{attribute 'reflection'} 
(* The VLT® PROFINET MCA 120 is used in combination with:
• VLT® HVAC Drive FC 102
• VLT® Refrigeration Drive FC 103
• VLT® AQUA Drive FC 202
• VLT® AutomationDrive FC 301/302
• VLT® Decentral Drive FCD 302
 *)
FUNCTION_BLOCK FB_Danfoss_VLT_MCA_120 EXTENDS FB_LinkDataReal
VAR_INPUT	
	stControl				: ST_Danfoss_VLT_MCA_120_Control;	
	stConfig 				: ST_Danfoss_VLT_MCA_120_Config;
END_VAR

VAR_OUTPUT
	stStatus				: ST_Danfoss_VLT_MCA_120_Status;
	fValue					: REAL;
END_VAR

VAR
    {attribute 'instance-path'} 
    {attribute 'noinit'} 
    sPath 					: STRING; 
	pFromBus				: POINTER TO BYTE;
	pToBus					: POINTER TO BYTE;	
	                    	
	fbProfidriveGSM			: FB_ProfidriveGSM;	
	fbMoveVelocity			: FB_MoveVelocity;
	
	fAcceleration	 		: REAL;
	fDeceleration		 	: REAL;
	fDecelerationQuickStop 	: REAL;
	fDecelerationCoastStop 	: REAL;
	bQuickStopExternal		: BOOL;
	
	bFaultPresent 			: BOOL;
	bAlarmPresent 			: BOOL;
	bInverterError 			: BOOL;
	bVoltageError 			: BOOL;
	bMomentError 			: BOOL;
	bTimerError 			: BOOL;
END_VAR

SUPER^();
InitRun();
ReadBus();
ControlLogic();
WriteBus();

(*Assign Process Data Objects to device*)
METHOD PUBLIC AssignProcessData : BOOL
VAR_INPUT
	aControlData 		: ANY; //Addr. Process Output (PO), 6 BYTES FROM FIELDBUS
	aStatusData 		: ANY; //Addr. Process Input (PI), 6 BYTES TO FIELDBUS
END_VAR
THIS^.pFromBus := aControlData.pValue;
THIS^.pToBus := aStatusData.pValue;
END_METHOD

METHOD INTERNAL ControlLogic
(* Evaluate/limit parameters *)
	EvaluateParameters();

(* Unity init - load position *)
	IF SUPER^.Status.7 THEN
		ControlData := StatusData;
	END_IF

(* Call base statemachine *)
fbProfidriveGSM.bStandstill						:= OC_Core.F_Compare(fbMoveVelocity.fVelocity, 0, 1E-3);
fbProfidriveGSM.stControl.b0_On 				:= stControl.bOFF1;
fbProfidriveGSM.stControl.b1_CoastStop 			:= stControl.bOFF2;
fbProfidriveGSM.stControl.b2_QuickStop 			:= stControl.bOFF3 AND NOT bQuickStopExternal;
fbProfidriveGSM.stControl.b3_EnableOperation	:= stControl.bEnableOperation;

(* Preset target values *)
	fbMoveVelocity.fTargetVelocity	:= 0;
	fbMoveVelocity.fAccMax 			:= fAcceleration;
	fbMoveVelocity.fDecMax 			:= fDeceleration;

(* Operation *)
	IF fbProfidriveGSM.eState = E_ProfidriveGSM_State.S4_Operation THEN	
		// Main setpoint
		IF NOT stControl.bJog1 AND NOT stControl.bJog2 THEN
			fbMoveVelocity.fTargetVelocity := (stControl.nSoll * stConfig.fP2000) / 16#4000;
		// Jog 1
		ELSIF stControl.bJog1 AND NOT stControl.bJog2 THEN
			fbMoveVelocity.fTargetVelocity := stConfig.fP1058;
		// Jog 2
		ELSIF NOT stControl.bJog1 AND stControl.bJog2 THEN	
			fbMoveVelocity.fTargetVelocity := stConfig.fP1059;
		END_IF
		
		// Stop
		IF NOT stControl.bOperatingCondition OR NOT stControl.bEnableSetpoint THEN
			fbMoveVelocity.fTargetVelocity := 0;
		END_IF
		
		// Reversing velocity
		IF stControl.bReversing THEN
			fbMoveVelocity.fTargetVelocity := -fbMoveVelocity.fTargetVelocity;
		END_IF
		
		// Hold velocity
		IF NOT stControl.bContinueRampFunctionGenerator AND NOT stControl.bJog1 AND NOT stControl.bJog2 THEN
			fbMoveVelocity.fTargetVelocity := fbMoveVelocity.fVelocity;
		END_IF	
		
	END_IF
	
(* Coast stop, Quick stop, Ramp stop *)
	IF fbProfidriveGSM.eState = E_ProfidriveGSM_State.S1_SwitchingOnInhibited THEN
		fbMoveVelocity.fTargetVelocity	:= 0;
		fbMoveVelocity.fAccMax 			:= fDecelerationCoastStop;
		fbMoveVelocity.fDecMax 			:= fDecelerationCoastStop;
	ELSIF fbProfidriveGSM.eState = E_ProfidriveGSM_State.S52_QuickStop THEN
		fbMoveVelocity.fTargetVelocity	:= 0;
		fbMoveVelocity.fAccMax 			:= fDecelerationQuickStop;
		fbMoveVelocity.fDecMax 			:= fDecelerationQuickStop;
	ELSIF fbProfidriveGSM.eState = E_ProfidriveGSM_State.S51_RampStop THEN
		fbMoveVelocity.fTargetVelocity	:= 0;
		fbMoveVelocity.fAccMax 			:= fDeceleration;
		fbMoveVelocity.fDecMax 			:= fDeceleration;
	END_IF

(* Call MoveVelocity *)
	fbMoveVelocity();
	
(* Status word *)
	stStatus.bReadyForSwitchingOn			:= fbProfidriveGSM.stStatus.b0_ReadyToSwitchOn;	
	stStatus.bReadyForOperation				:= fbProfidriveGSM.stStatus.b1_ReadyForOperation;
	stStatus.bOperationEnabled				:= stControl.bEnableOperation;
	stStatus.bFaultPresent					:= bFaultPresent;
	stStatus.bNoCoastDownActive				:= fbProfidriveGSM.eState <> E_ProfidriveGSM_State.S1_SwitchingOnInhibited;
	stStatus.bNoQuickStopActive				:= fbProfidriveGSM.eState <> E_ProfidriveGSM_State.S52_QuickStop;
	stStatus.bSwitchingOnInhibited			:= fbProfidriveGSM.stStatus.b6_SwitchingOnInhibited;
	stStatus.bAlarmPresent					:= bAlarmPresent;
	stStatus.bDeviationWithinTolerance		:= TRUE;
	stStatus.bControlRequested				:= stConfig.bControlRequested;	
	stStatus.bFrequencyLimitOk				:= TRUE;	
	stStatus.bBusy							:= ABS(fbMoveVelocity.fVelocity) > 0;
	stStatus.bInverterError					:= bInverterError;	
	stStatus.bVoltageError					:= bVoltageError;
	stStatus.bMomentError					:= bMomentError;
	stStatus.bTimerError					:= bTimerError;

(* Reset quickstop from extern *)
	IF stControl.bAcknowledgeFaults THEN
		bQuickStopExternal := FALSE;
	END_IF

(* Calculate NIST *)
	IF stConfig.fP2000 = 0 THEN
		stStatus.nIst	:= 0;
	ELSE
		stStatus.nIst	:=	REAL_TO_INT((ABS(fbMoveVelocity.fVelocity) * 16#4000) / stConfig.fP2000);
	END_IF

(* Output of actual value *)	
	IF stConfig.bOutputVelocity THEN
		ControlData := fbMoveVelocity.fVelocity;
	ELSE
		ControlData := ControlData + fbMoveVelocity.fVelocity *  GVL_Core.fbSystem.fDeltaTime * GVL_Core.fbSystem.fTimeScaling;
	END_IF
	
	fValue := ControlData;
END_METHOD

METHOD INTERNAL EvaluateParameters
VAR_INPUT
END_VAR
IF stConfig.fP1120 > 0 THEN
	fAcceleration := stConfig.fP2000/stConfig.fP1120;
ELSE
	fAcceleration := 1000;
END_IF

IF stConfig.fP1121 > 0 THEN
	fDeceleration := stConfig.fP2000/stConfig.fP1121;
ELSE
	fDeceleration := 1000;
END_IF

IF stConfig.fP1135 > 0 THEN
	fDecelerationQuickStop := stConfig.fP2000/stConfig.fP1135;
ELSE
	fDecelerationQuickStop := 1000;
END_IF

IF stConfig.fRampDownTimeCoastStop > 0 THEN
	fDecelerationCoastStop := stConfig.fP2000/stConfig.fRampDownTimeCoastStop;
ELSE
	fDecelerationCoastStop := 1000;
END_IF
END_METHOD

METHOD PUBLIC GetAcylicParameter : BOOL
VAR_INPUT
	stParameter : POINTER TO ST_PROFIdriveParam;
END_VAR
IF stParameter^.nNumber = 35 THEN
	stParameter^.nFormat := E_PROFIdriveParamFormat.FLOAT;
	stParameter^.nElements := 1;
	memcpy(ADR(stParameter^.aValue), ADR(stConfig.nR0035), 4);
END_IF
END_METHOD

METHOD INTERNAL InitRun : BOOL
VAR_INST
	bInitRun : BOOL := TRUE;
END_VAR
IF NOT bInitRun THEN RETURN; END_IF
bInitRun := FALSE;

IF pFromBus = 0 OR pToBus = 0 THEN
	ADSLOGSTR(ADSLOG_MSGTYPE_WARN, CONCAT(sPath, ': %s'), 'Plc address not set.');
END_IF
END_METHOD

METHOD INTERNAL ReadBus
VAR_INPUT
END_VAR
IF pFromBus = 0 THEN
	RETURN;
END_IF

IF NOT stConfig.bSwapProcessData THEN
	(* Control word *)
		stControl.bOFF1							:= pFromBus[0].0;
		stControl.bOFF2							:= pFromBus[0].1;
		stControl.bOFF3							:= pFromBus[0].2;
		stControl.bEnableOperation			    	:= pFromBus[0].3;
		stControl.bOperatingCondition				:= pFromBus[0].4;
		stControl.bContinueRampFunctionGenerator	:= pFromBus[0].5;
		stControl.bEnableSetpoint  				:= pFromBus[0].6;
		stControl.bAcknowledgeFaults				:= pFromBus[0].7;
		stControl.bJog1							:= pFromBus[1].0;
		stControl.bJog2							:= pFromBus[1].1;
		stControl.bDataValid						:= pFromBus[1].2;
		stControl.bFreqCorrDown					:= pFromBus[1].3;
		stControl.bFreqCorrUp						:= pFromBus[1].4;
		stControl.bParameterSelectionLSB			:= pFromBus[1].5;
		stControl.bParameterSelectionMSB			:= pFromBus[1].6;
		stControl.bReversing						:= pFromBus[1].7;
		
	(* Setpoint speed *)
		stControl.nSoll							:= UINT_TO_INT(pFromBus[2] + pFromBus[3] * 16#100);
ELSE
	(* Control word *)
		stControl.bOFF1							:= pFromBus[1].0;
		stControl.bOFF2							:= pFromBus[1].1;
		stControl.bOFF3							:= pFromBus[1].2;
		stControl.bEnableOperation				    := pFromBus[1].3;
		stControl.bOperatingCondition				:= pFromBus[1].4;
		stControl.bContinueRampFunctionGenerator	:= pFromBus[1].5;
		stControl.bEnableSetpoint  				:= pFromBus[1].6;
		stControl.bAcknowledgeFaults				:= pFromBus[1].7;
		stControl.bJog1							:= pFromBus[0].0;
		stControl.bJog2							:= pFromBus[0].1;
		stControl.bDataValid						:= pFromBus[0].2;
		stControl.bFreqCorrDown					:= pFromBus[0].3;
		stControl.bFreqCorrUp						:= pFromBus[0].4;
		stControl.bParameterSelectionLSB			:= pFromBus[0].5;
		stControl.bParameterSelectionMSB			:= pFromBus[0].6;
		stControl.bReversing						:= pFromBus[0].7;
		
	(* Setpoint speed *)
		stControl.nSoll							:= UINT_TO_INT(pFromBus[3] + pFromBus[2] * 16#100);
END_IF
END_METHOD

METHOD PUBLIC SetAcylicParameter : BOOL
VAR_INPUT
	pParameter : POINTER TO ST_PROFIdriveParam;
END_VAR
END_METHOD

METHOD PUBLIC TrigSafetyStop
bQuickStopExternal := TRUE;
END_METHOD

METHOD INTERNAL WriteBus
IF pToBus = 0 THEN
	RETURN;
END_IF

IF NOT stConfig.bSwapProcessData THEN
	(* Status word *)
		pToBus[0].0 := stStatus.bReadyForSwitchingOn			;	
		pToBus[0].1 := stStatus.bReadyForOperation				;
		pToBus[0].2 := stStatus.bOperationEnabled				;
		pToBus[0].3 := stStatus.bFaultPresent					;
		pToBus[0].4 := stStatus.bNoCoastDownActive				;
		pToBus[0].5 := stStatus.bNoQuickStopActive				;
		pToBus[0].6 := stStatus.bSwitchingOnInhibited			;
		pToBus[0].7 := stStatus.bAlarmPresent					;
		pToBus[1].0 := stStatus.bDeviationWithinTolerance		;
		pToBus[1].1 := stStatus.bControlRequested				;
		pToBus[1].2 := stStatus.bFrequencyLimitOk				;
		pToBus[1].3 := stStatus.bBusy							;
		pToBus[1].4 := stStatus.bInverterError 					;
		pToBus[1].5 := stStatus.bVoltageError					;	
		pToBus[1].6 := stStatus.bMomentError					;
		pToBus[1].7 := stStatus.bTimerError						;
	
	(* Actual speed *)
		memcpy(ADR(pToBus[3]), ADR(stStatus.nIst) + 1, 1);
		memcpy(ADR(pToBus[2]), ADR(stStatus.nIst), 1);
ELSE
	(* Status word *)
		pToBus[1].0 := stStatus.bReadyForSwitchingOn			;	
		pToBus[1].1 := stStatus.bReadyForOperation				;
		pToBus[1].2 := stStatus.bOperationEnabled				;
		pToBus[1].3 := stStatus.bFaultPresent					;
		pToBus[1].4 := stStatus.bNoCoastDownActive				;
		pToBus[1].5 := stStatus.bNoQuickStopActive				;
		pToBus[1].6 := stStatus.bSwitchingOnInhibited			;
		pToBus[1].7 := stStatus.bAlarmPresent					;
		pToBus[0].0 := stStatus.bDeviationWithinTolerance		;
		pToBus[0].1 := stStatus.bControlRequested				;
		pToBus[0].2 := stStatus.bFrequencyLimitOk				;
		pToBus[0].3 := stStatus.bBusy							;
		pToBus[0].4 := stStatus.bInverterError 					;
		pToBus[0].5 := stStatus.bVoltageError					;	
		pToBus[0].6 := stStatus.bMomentError					;
		pToBus[0].7 := stStatus.bTimerError						;
	
	(* Actual speed *)
		memcpy(ADR(pToBus[2]), ADR(stStatus.nIst) + 1, 1);
		memcpy(ADR(pToBus[3]), ADR(stStatus.nIst), 1);
END_IF
END_METHOD

END_FUNCTION_BLOCK

(* stored: Version 1.1.0.1, ProductVersion 3.1.4024.12
   POU FB_Danfoss_VLT_MCA_120: Id {33b5c3e5-e512-0435-183b-5e558dabb81d}, SpecialFunc None
   Method AssignProcessData: Id {8f82b332-a6ab-05b1-0554-5dd4ea1f4a7c}
   Method ControlLogic: Id {bac93425-3673-063e-0f09-d78825a2fc8d}
   Method EvaluateParameters: Id {512947c7-6289-09b6-3f77-c699010fa861}
   Method GetAcylicParameter: Id {2cdb7e82-6639-0168-114d-4e1ad369c456}
   Method InitRun: Id {920237f5-c729-0104-3b82-f9c2379f2a07}
   Method ReadBus: Id {398713c8-c7cb-00d4-02d0-3195f493fbf6}
   Method SetAcylicParameter: Id {4634cec4-9032-0784-0b07-40e999b37e5b}
   Method TrigSafetyStop: Id {360c40e5-a457-033d-2436-9ea2232f2b24}
   Method WriteBus: Id {b2dbeac5-6f3b-0239-3f5a-8ff3fd92f963} *)
